{attribute 'linkalways'} 
{attribute 'no_explicit_call' := 'This FB is a CLASS and must be accessed using methods or properties'}
{attribute 'enable_dynamic_creation'}
FUNCTION_BLOCK _ETcVnFilterDirection EXTENDS EnumDatatypeBase
VAR
	localData : ETcVnFilterDirection;
	activeData : REFERENCE TO ETcVnFilterDirection;
	enumBaseDatatype : _INT(localData);
END_VAR

METHOD PRIVATE AddLocalEnumeration
VAR_INPUT
	Enumeration : T_MAXSTRING;
	Value : ETcVnFilterDirection;
END_VAR
AddEnumeration(Enumeration, Value);
END_METHOD

PROPERTY PUBLIC Address : PVOID
GET
Address := ADR(activeData);
END_GET
END_PROPERTY

METHOD PUBLIC ClearReference
VAR_INPUT
END_VAR
activeData REF= localData;
SetBaseDatatypeReference();
END_METHOD

METHOD PUBLIC Clone : I_Datatype
VAR
    pClone : POINTER TO _ETcVnFilterDirection;
END_VAR
pClone := __NEW(_ETcVnFilterDirection(InitialValue := Value));
Clone := pClone^;
END_METHOD

METHOD FB_init : BOOL
VAR_INPUT
	bInitRetains : BOOL; // if TRUE, the retain variables are initialized (warm start / cold start)
	bInCopyCode : BOOL;  // if TRUE, the instance afterwards gets moved into the copy code (online change)
	InitialValue : ETcVnFilterDirection;
END_VAR
localData := InitialValue;
AddBaseDatatype(enumBaseDatatype);
ClearReference();

AddLocalEnumeration('TCVN_FD_X', ETcVnFilterDirection.TCVN_FD_X);
AddLocalEnumeration('TCVN_FD_Y', ETcVnFilterDirection.TCVN_FD_Y);
END_METHOD

PROPERTY PUBLIC Identifier : T_MAXSTRING
GET
Identifier := 'ETcVnFilterDirection';
END_GET
END_PROPERTY

METHOD IsEnumeratorValueEqual : BOOL
VAR_INPUT
	Enumerator : I_KeyValueForwardEnumerator;
END_VAR
VAR
	storedValue : ETcVnFilterDirection;
END_VAR
IF NOT Enumerator.TryGet(storedValue) THEN
	RETURN;
END_IF

IsEnumeratorValueEqual := storedValue = activeData;
END_METHOD

METHOD PUBLIC MakeReferenceTo
VAR_INPUT
	ReferenceTarget : REFERENCE TO ETcVnFilterDirection;
END_VAR
activeData REF= ReferenceTarget;
SetBaseDatatypeReference();
END_METHOD

METHOD PROTECTED SetBaseDatatypeReference
VAR_INPUT
END_VAR
enumBaseDatatype.MakeReferenceTo(activeData);
END_METHOD

PROPERTY PUBLIC Size : UDINT
GET
Size := SIZEOF(activeData);
END_GET
END_PROPERTY

METHOD TryMakeReferenceTo : BOOL
VAR_INPUT
	Target : I_Datatype;
END_VAR
VAR
	targetAsEnum : I_EnumDatatype;
	pTargetData : POINTER TO ETcVnFilterDirection;
END_VAR
IF NOT Target.TryResolveAsEnumDatatype(targetAsEnum) THEN
	RETURN;
END_IF

IF targetAsEnum.Identifier <> Identifier THEN
	RETURN;
END_IF

pTargetData := Target.Address;
activeData REF= pTargetData^;
SetBaseDatatypeReference();
TryMakeReferenceTo := TRUE;
END_METHOD

PROPERTY PUBLIC Value : ETcVnFilterDirection
GET
Value := activeData;
END_GET
SET
activeData := Value;
END_SET
END_PROPERTY

END_FUNCTION_BLOCK

(* stored: Version 1.1.0.1, ProductVersion 3.1.4024.12
   POU _ETcVnFilterDirection: Id {01e13ddb-971f-4193-8a73-a1e40492dfa0}, SpecialFunc None
   Folder Constructor: Id {65370781-2964-4c94-a1a7-84c4339bb9e0}
   Folder Private: Id {7945db41-649b-4545-8ede-17e9e710ba93}
   Folder Protected: Id {69450e07-1729-454b-8d0b-4ba3f69f5316}
   Method AddLocalEnumeration: Id {baf2c460-56c4-419e-9526-93341b776902}
   Property Address: Id {1c8def0f-e8f7-4c3e-bfb1-98c111d17220}
   Get Get: Id {81471561-c312-47ad-a8f0-31e2efd33849}
   Method ClearReference: Id {f8dc53d3-17c5-4e00-aa92-69a52c38990e}
   Method Clone: Id {a2405b3d-1a0b-4404-b36e-00cea760c9df}
   Method FB_init: Id {d32a624f-080d-4222-9ec1-d16b8b863ab5}
   Property Identifier: Id {fdedb157-90b7-437c-8fc3-e902de16ad6e}
   Get Get: Id {a25f379b-3d02-4016-baef-2469761de5f3}
   Method IsEnumeratorValueEqual: Id {f7faffd3-bd37-47db-804e-0c0930b4cba9}
   Method MakeReferenceTo: Id {72a504de-2364-4991-97f9-157e8738824c}
   Method SetBaseDatatypeReference: Id {965d6d1e-6dd6-41e3-8b8a-57df1f16f50e}
   Property Size: Id {f1ae10e0-fa19-4bde-897b-cd4ada9807b3}
   Get Get: Id {c33a3ae8-5eaa-4d6a-ab08-56cb948c619d}
   Method TryMakeReferenceTo: Id {02871e57-2a9b-48b8-9b92-4e39fe400903}
   Property Value: Id {5b852f04-d3b0-44e0-b6a5-5d0a59a17a7f}
   Get Get: Id {44f4880f-e1d6-4330-9833-e293c9929354}
   Set Set: Id {16a3e01a-d52d-4321-9f41-95689b2cf46b} *)
